{attribute 'qualified_only'}
VAR_GLOBAL
	Coil : ARRAY[1..10] OF ST_Recipe;
	General : ST_Recipe;
END_VAR

(* stored: Version 1.1.0.1, ProductVersion 3.1.4024.11
   GVL Recipe: Id {76a52482-bd91-4c6a-bc62-c12593ed89ca} *)
